TYPE ST_Output :
STRUCT
	xBusy: BOOL;
	xError: BOOL;
	nErrID : INT;
	Resulte : STRING;
	Resulth : STRING;
	Resultd : STRING;
	Boole : INT;
	Boolh : INT;
	Boold : INT;
END_STRUCT
END_TYPE

(* stored: Version 1.1.0.1, ProductVersion 3.1.4020.6
   DUT ST_Output: Id {00b1120f-c2a9-4e00-b1c1-eac632684d1a} *)
